// TwinCAT 3 PLC project StateCtrl
// ProgramVersion: 3.1.4026.1+c9eadab3edd020c56c333d811d5b3c408c2550c8
// CompilerDefines: VISU_USEPROPERTYINFO
// libraries:
//   Tc2_Standard, * (Beckhoff Automation GmbH)
//   Tc2_System, * (Beckhoff Automation GmbH)
//   VisuSymbols, 4.5.0.0 (System)
// project tree:
//   / GlobalTextList.TcGTLO, PlcTask.TcTTO, Visualization Manager.TcVMO (not stored), VISU_TASK.TcTTO
//   GVLs/ Indicator.TcGVL, Input.TcGVL, MR_J_Motor.TcGVL, SignalOut.TcGVL
//   POUs/ MAIN.TcPOU, POU_1.TcPOU
//   VISUs/ Visualization_reference.TcVIS
// real-time tasks:
//   TASK PlcTask: cycle T#10ms, priority 20, ADS port 350
//   TASK VISU_TASK: cycle T#200000us, priority 30, ADS port 351
// I/O:
//   DEVICE Device 1 (EtherCAT), AmsNetId 192.168.5.28.2.1
//     Term 1 (EK1828) [EK1828 EtherCAT IO-Coupler  (1A E-Bus, 4 Ch. Dig. In, 3ms, 8 Ch. Dig. Out 24V, 0,5A)]
//     Term 2 (EK1100) [EK1100 EtherCAT Coupler (2A E-Bus)]
//       Term 3 (EL1889) [EL1889 16Ch. Dig. Input 24V, 3ms, negative]
//       Term 4 (EL2889) [EL2889 16Ch. Dig. Output 24V, 0.5A, negative]
//       Term 5 (EL4002) [EL4002 2Ch. Ana. Output 0-10V, 12bit]
//       Term 6 (EL5101) [EL5101 1Ch. Inc. Encoder 5V]
//       Term 7 (EL9011) [EL9011 End Terminal]
// variable links:
//   StateCtrl/StateCtrl Instance <-> Device 1 (EtherCAT)/Term 1 (EK1828)
//     PlcTask Inputs/Input.bEMG <-> Channel 3/Input
//     PlcTask Inputs/Input.bEnable <-> Channel 1/Input
//     PlcTask Inputs/Input.bSWGreen <-> Channel 4/Input
//     PlcTask Inputs/Input.bSWRed <-> Channel 2/Input
//     PlcTask Outputs/Indicator.bSWGreen <-> Channel 7/Output
//     PlcTask Outputs/Indicator.bSWRed <-> Channel 5/Output
//     PlcTask Outputs/SignalOut.bStart <-> Channel 6/Output
//   StateCtrl/StateCtrl Instance <-> Device 1 (EtherCAT)/Term 2 (EK1100)/Term 4 (EL2889)
//     PlcTask Outputs/MR_J_Motor.bCCW <-> Channel 3/Output
//     PlcTask Outputs/MR_J_Motor.bCW <-> Channel 2/Output
//     PlcTask Outputs/MR_J_Motor.bReset <-> Channel 4/Output
//     PlcTask Outputs/MR_J_Motor.bSON <-> Channel 1/Output
//   StateCtrl/StateCtrl Instance <-> Device 1 (EtherCAT)/Term 2 (EK1100)/Term 5 (EL4002)
//     PlcTask Outputs/MR_J_Motor.iInVoltage <-> AO Outputs Channel 1/Analog output

CONFIGURATION StateCtrl
    RESOURCE PLC ON TwinCAT3
        TASK PlcTask(INTERVAL := T#10ms, PRIORITY := 20);
        TASK VISU_TASK(INTERVAL := T#200000us, PRIORITY := 30);
        PROGRAM MAIN WITH PlcTask : MAIN;
        PROGRAM POU_1 WITH PlcTask : POU_1;
        PROGRAM VisuElems_Visu_Prg WITH VISU_TASK : VisuElems.Visu_Prg;
    END_RESOURCE
END_CONFIGURATION

// ---- GVLs/Indicator.TcGVL
{attribute 'qualified_only'}
VAR_GLOBAL
	bSWGreen 	AT%Q*	:BOOL;
	bSWRed 		AT%Q*	:BOOL;
END_VAR

// ---- GVLs/Input.TcGVL
{attribute 'qualified_only'}
VAR_GLOBAL
	bEMG 		AT%I*	:BOOL;
	bEnable 	AT%I*	:BOOL;
	bSWGreen 	AT%I*	:BOOL;
	bSWRed 		AT%I*	:BOOL;
	iHMISlide: INT;
END_VAR

// ---- GVLs/MR_J_Motor.TcGVL
{attribute 'qualified_only'}
VAR_GLOBAL
	bReset 		AT%Q*	:BOOL;
	bSON 		AT%Q*	:BOOL;
	bCW 		AT%Q*	:BOOL;
	bCCW 		AT%Q*	:BOOL;
	iInVoltage  AT%Q*	:INT;
END_VAR

// ---- GVLs/SignalOut.TcGVL
{attribute 'qualified_only'}
VAR_GLOBAL
	bStart AT%Q*	:BOOL;
END_VAR

// ---- POUs/MAIN.TcPOU
PROGRAM MAIN
VAR
END_VAR

END_PROGRAM

// ---- POUs/POU_1.TcPOU
PROGRAM POU_1
VAR
	T0: TOF;
	Te: TIME;
END_VAR

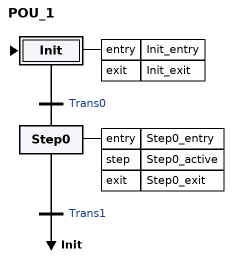
INITIAL_STEP Init:
    Init_entry(P1);  // entry action
    Init_exit(P0);  // exit action
END_STEP
TRANSITION FROM Init TO Step0
    := Trans0;
END_TRANSITION
STEP Step0:
    Step0_entry(P1);  // entry action
    Step0_active(N);  // step action
    Step0_exit(P0);  // exit action
END_STEP
TRANSITION FROM Step0 TO Init
    := Trans1;
END_TRANSITION

ACTION Init_entry:
Indicator.bSWGreen := TRUE;
SignalOut.bStart := TRUE;
END_ACTION

ACTION Init_exit:
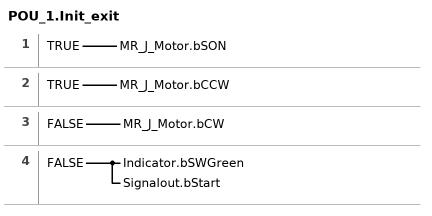
// NETWORK 1
MR_J_Motor.bSON := TRUE;

// NETWORK 2
MR_J_Motor.bCCW := TRUE;

// NETWORK 3
MR_J_Motor.bCW := FALSE;

// NETWORK 4
Indicator.bSWGreen := FALSE;
Signalout.bStart := FALSE;
END_ACTION

ACTION Step0_active:
Indicator.bSWGreen:=T0.Q;
Te := T0.ET;

IF Input.iHMISlide >= 0THEN
	MR_J_Motor.bCW := TRUE;
	MR_J_Motor.bCCW := FALSE;
ELSE
	MR_J_Motor.bCW := FALSE;
	MR_J_Motor.bCCW := TRUE;
END_IF
MR_J_Motor.iInVoltage := ABS(Input.iHMISlide);
END_ACTION

ACTION Step0_entry:
Indicator.bSWRed := TRUE;
END_ACTION

ACTION Step0_exit:
Indicator.bSWRed := FALSE;
MR_J_Motor.bSON := FALSE;
END_ACTION

TRANSITION Trans0:
Trans0:= (NOT Input.bSWGreen) AND Input.bEnable;
END_TRANSITION

TRANSITION Trans1:
Trans1 := (NOT Input.bSWRed) OR (NOT Input.bEMG);
END_TRANSITION

END_PROGRAM

// ---- GlobalTextList.TcGTLO
TEXTLIST GlobalTextList
  318 = 'CCW'
  97 = 'CW'
  838 = 'Motor Input'
END_TEXTLIST

// ---- VISUs/Visualization_reference.TcVIS
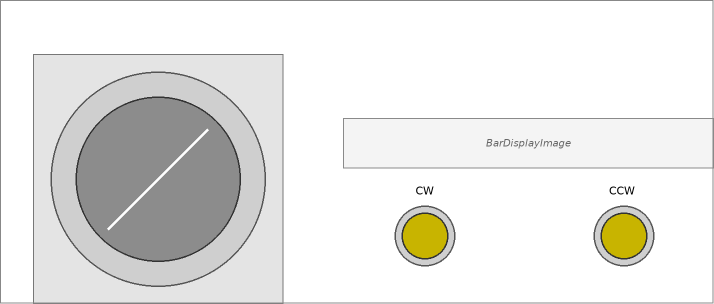
VISUALIZATION Visualization_reference  // 714x304
    Potentiometer360 (33,54 250x250), variable: Input.iHMISlide, style: Potentiometer-Potentiometer360-Gray, scale format: %.1f, scale -660..660
        p2431819421: Outside
    BarDisplayImage (343,118 371x50), value: MR_J_Motor.iInVoltage, style: BarDisplayImage-Gray, scale format: %.1f, scale 0..660
    Lamp1 (390,201 70x70), variable: MR_J_Motor.bCW, style: Lamp-Lamp1-Yellow
    Lamp1 (589,201 70x70), variable: MR_J_Motor.bCCW, style: Lamp-Lamp1-Yellow
    Label (350,176 150x30), "CW"
    Label (547,176 150x30), "CCW"
END_VISUALIZATION
